Omron Sysmac Studio project DEMO_10 (Sysmac Studio 1.45.1.64010, StandardProject)

# Controller PLC: NX1P2-9024DT1 version 1.40
Task PrimaryTask (priority 4, period or condition 2000): Main_Prg
Library Mekatronik 1.0.0 (contents left out)

TYPE unW : UNION
    B : ARRAY[0..15] OF BOOL;
    BYT : ARRAY[0..1] OF BYTE;
    W : WORD;
END_UNION END_TYPE
TYPE unAlarm : UNION
    B : ARRAY[0..127] OF BOOL;
    LW : ARRAY[0..1] OF LWORD;
END_UNION END_TYPE
TYPE unUyari : UNION
    B : ARRAY[0..127] OF BOOL;
    LW : ARRAY[0..1] OF LWORD;
END_UNION END_TYPE
TYPE unTest : UNION
    B : ARRAY[0..127] OF BOOL;
    LW : ARRAY[0..1] OF LWORD;
END_UNION END_TYPE
TYPE ePLC_IO_St : STRUCT
    RealVars : ARRAY[1..64] OF REAL;  (* offset 0.0 *)
    IntegerVars : ARRAY[1..24] OF INT;  (* offset 256.0 *)
    String1_length : DINT;  (* offset 304.0 *)
    String1Var : STRING[82];  (* offset 308.0 *)
    String2_length : DINT;  (* offset 392.0 *)
    String2Var : STRING[82];  (* offset 396.0 *)
    SignalVars : ARRAY[1..64] OF BOOL;  (* offset 480.0 *)
END_STRUCT END_TYPE

VAR_GLOBAL
    From_Robot_C1 : ePLC_IO_St;  (* network input *)
    To_Robot_C1 : ePLC_IO_St;  (* network output *)
END_VAR

PROGRAM Main_Prg
VAR
    ToRo_Satrt : BOOL;
    FromRo_RobotAutoMode : BOOL;
    ytujty : REAL;
    ToRo_HareketModu : REAL;
    ToRo_IndexNumber : REAL;
    ToRo_PaletKat : REAL;
    FromRo_Haberlesme : BOOL;
    ToRo_Haberlesme : BOOL;
    konum_ok : BOOL;
    ToRo_x : REAL;
    ToRo_y : REAL;
    ToRo_z : REAL;
    ToRo_yaw : REAL;
    ToRo_pitch : REAL;
    ToRo_roll : REAL;
    izin : BOOL;
    ok : BOOL;
    campos : BOOL;
    campos1 : BOOL;
    konum1_ok : BOOL;
    ToRo_x1 : REAL;
    ToRo_y1 : REAL;
    ToRo_z1 : REAL;
    ToRo_yaw1 : REAL;
    ToRo_pitch1 : REAL;
    ToRo_roll1 : REAL;
END_VAR
VAR_EXTERNAL
    From_Robot_C1 : ePLC_IO_St;
    To_Robot_C1 : ePLC_IO_St;
END_VAR
VAR
    _e1 : R_TRIG;
    _e2 : R_TRIG;
    _e3 : R_TRIG;
    _e4 : R_TRIG;
END_VAR

(* Section Genel: ladder, written here as Structured Text *)

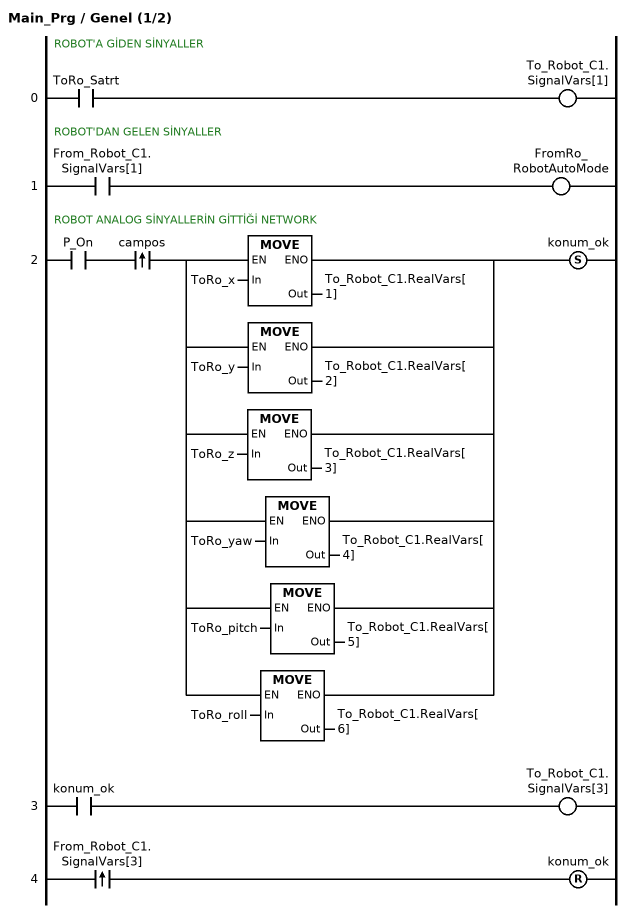
(* Rung 0: ROBOT'A GİDEN SİNYALLER *)
To_Robot_C1.SignalVars[1] := ToRo_Satrt;
(* Rung 1: ROBOT'DAN GELEN SİNYALLER *)
FromRo_RobotAutoMode := From_Robot_C1.SignalVars[1];
(* Rung 2: ROBOT ANALOG SİNYALLERİN GİTTİĞİ NETWORK *)
_e1(CLK := campos);
IF P_On AND _e1.Q THEN
    To_Robot_C1.RealVars[1] := ToRo_x;
    To_Robot_C1.RealVars[2] := ToRo_y;
    To_Robot_C1.RealVars[3] := ToRo_z;
    To_Robot_C1.RealVars[4] := ToRo_yaw;
    To_Robot_C1.RealVars[5] := ToRo_pitch;
    To_Robot_C1.RealVars[6] := ToRo_roll;
    konum_ok := TRUE;
END_IF;
(* Rung 3 *)
To_Robot_C1.SignalVars[3] := konum_ok;
(* Rung 4 *)
_e2(CLK := From_Robot_C1.SignalVars[3]);
IF _e2.Q THEN konum_ok := FALSE; END_IF;

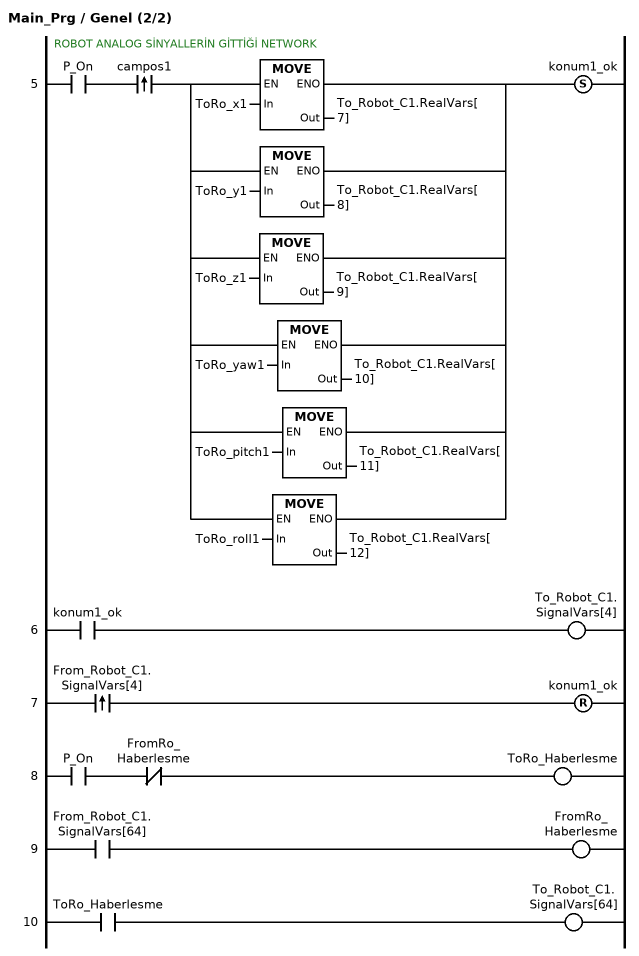
(* Rung 5: ROBOT ANALOG SİNYALLERİN GİTTİĞİ NETWORK *)
_e3(CLK := campos1);
IF P_On AND _e3.Q THEN
    To_Robot_C1.RealVars[7] := ToRo_x1;
    To_Robot_C1.RealVars[8] := ToRo_y1;
    To_Robot_C1.RealVars[9] := ToRo_z1;
    To_Robot_C1.RealVars[10] := ToRo_yaw1;
    To_Robot_C1.RealVars[11] := ToRo_pitch1;
    To_Robot_C1.RealVars[12] := ToRo_roll1;
    konum1_ok := TRUE;
END_IF;
(* Rung 6 *)
To_Robot_C1.SignalVars[4] := konum1_ok;
(* Rung 7 *)
_e4(CLK := From_Robot_C1.SignalVars[4]);
IF _e4.Q THEN konum1_ok := FALSE; END_IF;
(* Rung 8 *)
ToRo_Haberlesme := P_On AND NOT FromRo_Haberlesme;
(* Rung 9 *)
FromRo_Haberlesme := From_Robot_C1.SignalVars[64];
(* Rung 10 *)
To_Robot_C1.SignalVars[64] := ToRo_Haberlesme;
END_PROGRAM

FUNCTION_BLOCK myHome_FB
VAR
    MC_SetPosition_Homming : MC_SetPosition;
    MC_MoveAbsolute_Homming : MC_MoveAbsolute;
    Step_Home : INT;
    MC_MoveVelocity_1 : MC_MoveVelocity;
    TON_5 : TON;
    TON_6 : TON;
    MC_MoveVelocity_2 : MC_MoveVelocity;
    MC_MoveVelocity_11 : MC_MoveVelocity;
    MC_MoveVelocity_12 : MC_MoveVelocity;
    TP_1 : TP;
    TON_1 : TON;
    TON_2 : TON;
    Stop_Axis_1 : BOOL;
    Stop_Axis_2 : BOOL;
    HomePositionSensorInternal : LREAL;
    MC_Stop_Homming1 : MC_Stop;
    MC_Stop_Homming2 : MC_Stop;
    InPlaceHomed : BOOL;
    tr : BOOL;
    tr1 : BOOL;
END_VAR
VAR_IN_OUT CONSTANT
    Axis : _sAXIS_REF;
END_VAR
VAR_INPUT
    Start_Homming : BOOL;
    Direction : BOOL;
    ReverseDown : BOOL;
    UP_DN : BOOL;
    InPlace : BOOL;
    Home_Sensor : BOOL;
    EMG : BOOL;
    Stop : BOOL;
    HomeSpeed : LREAL;
    HomeSpeedLow : LREAL;
    OffsetPosition : LREAL;
    HomeSensorPosition : LREAL;
    ResetHomeOK : BOOL;
    IleriLimit : BOOL;
    GeriLimit : BOOL;
    Acceleration : LREAL;
    Deceleration : LREAL;
END_VAR
VAR_OUTPUT
    Home_Ok : BOOL;
    Busy : BOOL;
    Error : BOOL;
    LimitsError : BOOL;
END_VAR
VAR
    _e1 : R_TRIG;
    _p2 : BOOL;
    _p3 : BOOL;
    _br13_0 : BOOL;
    _br13_1 : BOOL;
    _br13_2 : BOOL;
    _e4 : R_TRIG;
    _e5 : R_TRIG;
    _e6 : R_TRIG;
    _e7 : F_TRIG;
    _br17_0 : BOOL;
    _br17_1 : BOOL;
    _br17_2 : BOOL;
    _e8 : R_TRIG;
END_VAR
(* ladder, written here as Structured Text *)

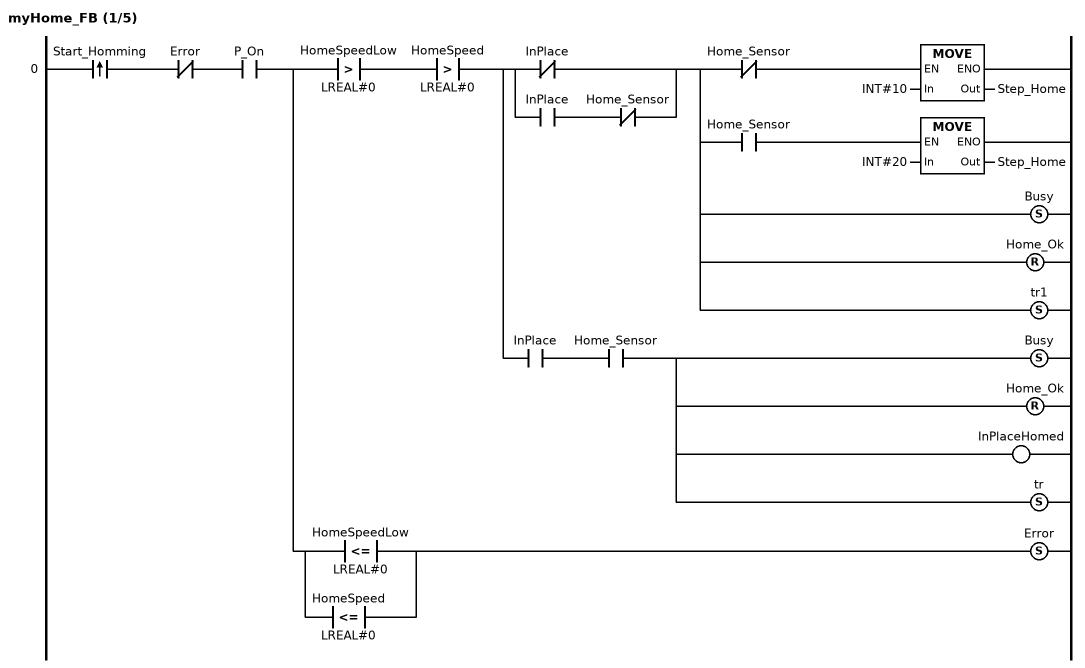
(* Rung 0 *)
_e1(CLK := Start_Homming);
_p2 := _e1.Q AND NOT Error AND P_On AND (HomeSpeedLow > LREAL#0) AND (HomeSpeed > LREAL#0);
_p3 := _p2 AND (NOT InPlace OR (InPlace AND NOT Home_Sensor));
IF _p3 AND NOT Home_Sensor THEN Step_Home := INT#10; END_IF;
IF _p3 AND Home_Sensor THEN Step_Home := INT#20; END_IF;
IF _p3 THEN
    Busy := TRUE;
    Home_Ok := FALSE;
    tr1 := TRUE;
END_IF;
IF _p2 AND InPlace AND Home_Sensor THEN
    Busy := TRUE;
    Home_Ok := FALSE;
END_IF;
InPlaceHomed := _p2 AND InPlace AND Home_Sensor;
IF _p2 AND InPlace AND Home_Sensor THEN tr := TRUE; END_IF;
IF _e1.Q AND NOT Error AND P_On AND ((HomeSpeedLow <= LREAL#0) OR (HomeSpeed <= LREAL#0)) THEN
    Error := TRUE;
END_IF;

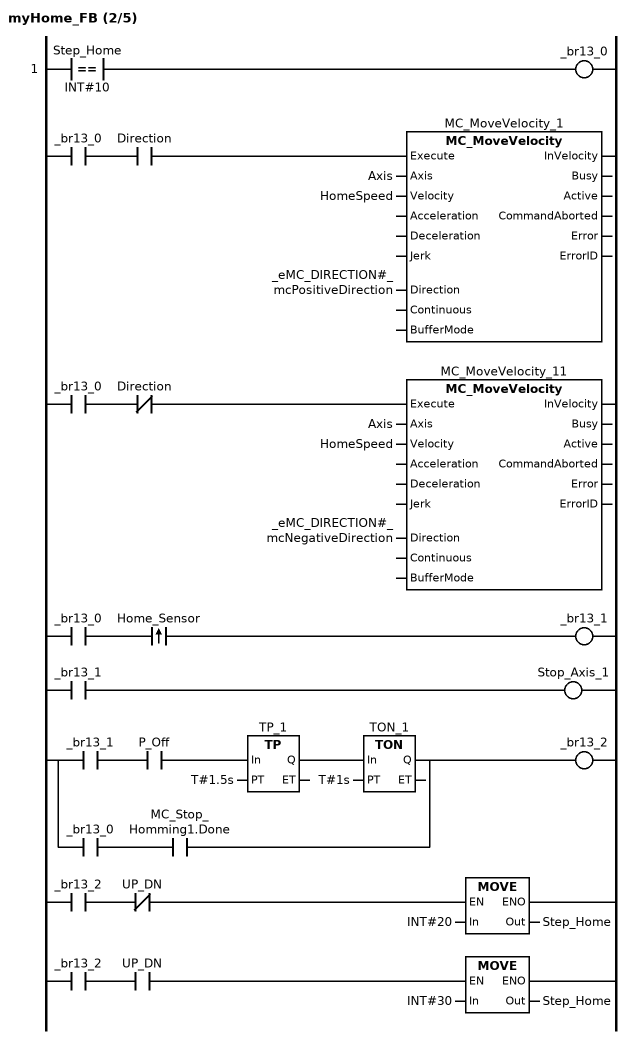
(* Rung 1 *)
_br13_0 := Step_Home = INT#10;
MC_MoveVelocity_1(Execute := _br13_0 AND Direction, Axis := Axis, Velocity := HomeSpeed, Direction := _eMC_DIRECTION#_mcPositiveDirection);
MC_MoveVelocity_11(Execute := _br13_0 AND NOT Direction, Axis := Axis, Velocity := HomeSpeed, Direction := _eMC_DIRECTION#_mcNegativeDirection);
_e4(CLK := Home_Sensor);
_br13_1 := _br13_0 AND _e4.Q;
Stop_Axis_1 := _br13_1;
TP_1(In := _br13_1 AND P_Off, PT := T#1.5s);
TON_1(In := TP_1.Q, PT := T#1s);
_br13_2 := TON_1.Q OR (_br13_0 AND MC_Stop_Homming1.Done);
IF _br13_2 AND NOT UP_DN THEN Step_Home := INT#20; END_IF;
IF _br13_2 AND UP_DN THEN Step_Home := INT#30; END_IF;

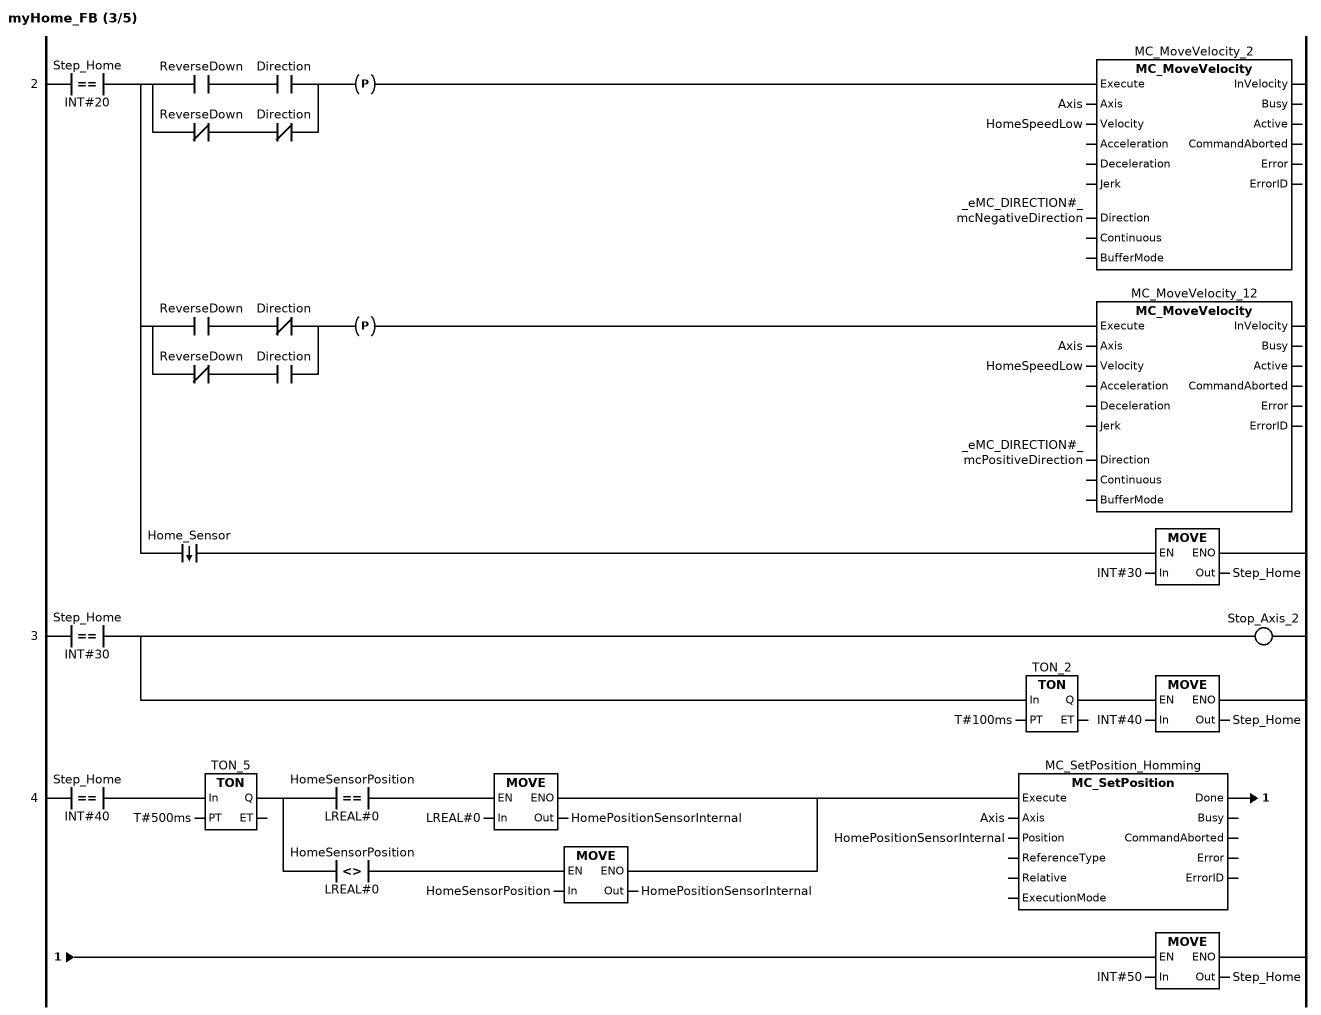
(* Rung 2 *)
_e5(CLK := (Step_Home = INT#20) AND ((ReverseDown AND Direction) OR (NOT ReverseDown AND NOT Direction)));
MC_MoveVelocity_2(Execute := _e5.Q, Axis := Axis, Velocity := HomeSpeedLow, Direction := _eMC_DIRECTION#_mcNegativeDirection);
_e6(CLK := (Step_Home = INT#20) AND ((ReverseDown AND NOT Direction) OR (NOT ReverseDown AND Direction)));
MC_MoveVelocity_12(Execute := _e6.Q, Axis := Axis, Velocity := HomeSpeedLow, Direction := _eMC_DIRECTION#_mcPositiveDirection);
_e7(CLK := Home_Sensor);
IF (Step_Home = INT#20) AND _e7.Q THEN Step_Home := INT#30; END_IF;
(* Rung 3 *)
Stop_Axis_2 := Step_Home = INT#30;
TON_2(In := Step_Home = INT#30, PT := T#100ms);
IF TON_2.Q THEN Step_Home := INT#40; END_IF;
(* Rung 4 *)
TON_5(In := Step_Home = INT#40, PT := T#500ms);
IF TON_5.Q AND (HomeSensorPosition = LREAL#0) THEN HomePositionSensorInternal := LREAL#0; END_IF;
IF TON_5.Q AND (HomeSensorPosition <> LREAL#0) THEN
    HomePositionSensorInternal := HomeSensorPosition;
END_IF;
MC_SetPosition_Homming(Execute := TON_5.Q AND ((HomeSensorPosition = LREAL#0) OR (HomeSensorPosition <> LREAL#0)), Axis := Axis, Position := HomePositionSensorInternal);
IF MC_SetPosition_Homming.Done THEN Step_Home := INT#50; END_IF;

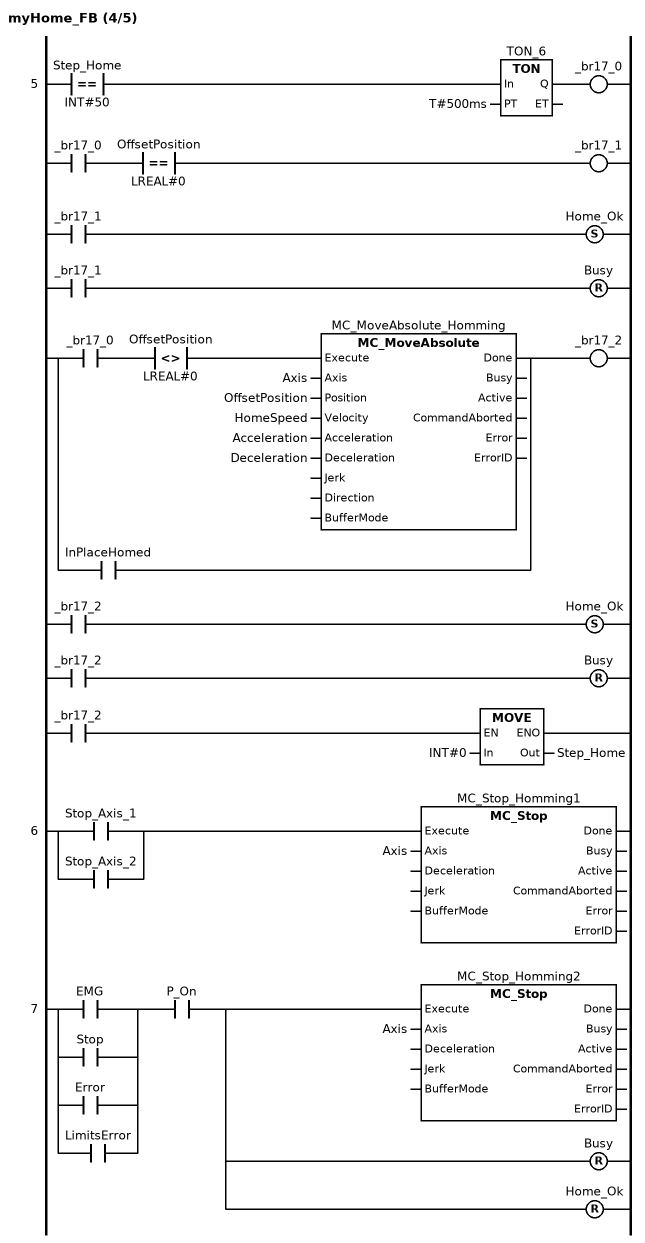
(* Rung 5 *)
TON_6(In := Step_Home = INT#50, PT := T#500ms);
_br17_0 := TON_6.Q;
_br17_1 := _br17_0 AND (OffsetPosition = LREAL#0);
IF _br17_1 THEN Home_Ok := TRUE; END_IF;
IF _br17_1 THEN Busy := FALSE; END_IF;
MC_MoveAbsolute_Homming(Execute := _br17_0 AND (OffsetPosition <> LREAL#0), Axis := Axis, Position := OffsetPosition, Velocity := HomeSpeed, Acceleration := Acceleration, Deceleration := Deceleration);
_br17_2 := MC_MoveAbsolute_Homming.Done OR InPlaceHomed;
IF _br17_2 THEN Home_Ok := TRUE; END_IF;
IF _br17_2 THEN Busy := FALSE; END_IF;
IF _br17_2 THEN Step_Home := INT#0; END_IF;
(* Rung 6 *)
MC_Stop_Homming1(Execute := Stop_Axis_1 OR Stop_Axis_2, Axis := Axis);
(* Rung 7 *)
MC_Stop_Homming2(Execute := (EMG OR Stop OR Error OR LimitsError) AND P_On, Axis := Axis);
IF (EMG OR Stop OR Error OR LimitsError) AND P_On THEN
    Busy := FALSE;
    Home_Ok := FALSE;
END_IF;

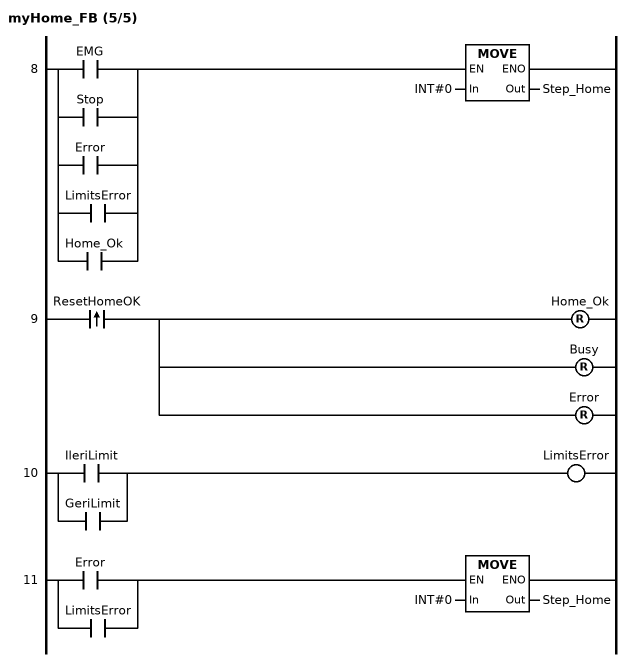
(* Rung 8 *)
IF EMG OR Stop OR Error OR LimitsError OR Home_Ok THEN Step_Home := INT#0; END_IF;
(* Rung 9 *)
_e8(CLK := ResetHomeOK);
IF _e8.Q THEN
    Home_Ok := FALSE;
    Busy := FALSE;
    Error := FALSE;
END_IF;
(* Rung 10 *)
LimitsError := IleriLimit OR GeriLimit;
(* Rung 11 *)
IF Error OR LimitsError THEN Step_Home := INT#0; END_IF;
END_FUNCTION_BLOCK

FUNCTION_BLOCK myHomeV2_FB
VAR
    MC_SetPosition_Homming : MC_SetPosition;
    MC_MoveAbsolute_Homming : MC_MoveAbsolute;
    Step_Home : INT;
    MC_MoveVelocity_1 : MC_MoveVelocity;
    TON_6 : TON;
    MC_MoveVelocity_2 : MC_MoveVelocity;
    MC_MoveVelocity_11 : MC_MoveVelocity;
    MC_MoveVelocity_12 : MC_MoveVelocity;
    TON_1 : TON;
    Stop_Axis_1 : BOOL;
    Stop_Axis_2 : BOOL;
    HomePositionSensorInternal : LREAL;
    MC_Stop_Homming1 : MC_Stop;
    MC_Stop_Homming2 : MC_Stop;
    InPlaceHomed : BOOL;
    Stop_Axis_Done : BOOL;
    Busy1 : BOOL;
    Busy2 : BOOL;
END_VAR
VAR_IN_OUT CONSTANT
    Axis : _sAXIS_REF;
END_VAR
VAR_INPUT
    Start_Homming : BOOL;
    Direction : BOOL;
    ReverseDown : BOOL;
    UP_DN : BOOL;
    InPlace : BOOL;
    Home_Sensor : BOOL;
    EMG : BOOL;
    Stop : BOOL;
    HomeSpeed : LREAL;
    HomeSpeedLow : LREAL;
    OffsetPosition : LREAL;
    HomeSensorPosition : LREAL;
    ResetHomeOK : BOOL;
    IleriLimit : BOOL;
    GeriLimit : BOOL;
    Acceleration : LREAL;
    Deceleration : LREAL;
END_VAR
VAR_OUTPUT
    Home_Ok : BOOL;
    Busy : BOOL;
    Error : BOOL;
    LimitsError : BOOL;
END_VAR
VAR
    _e1 : R_TRIG;
    _p2 : BOOL;
    _p3 : BOOL;
    _e4 : R_TRIG;
    _e5 : R_TRIG;
    _p6 : BOOL;
    _e7 : F_TRIG;
    _br30_0 : BOOL;
    _br30_1 : BOOL;
    _br30_2 : BOOL;
    _e8 : R_TRIG;
END_VAR
(* ladder, written here as Structured Text *)

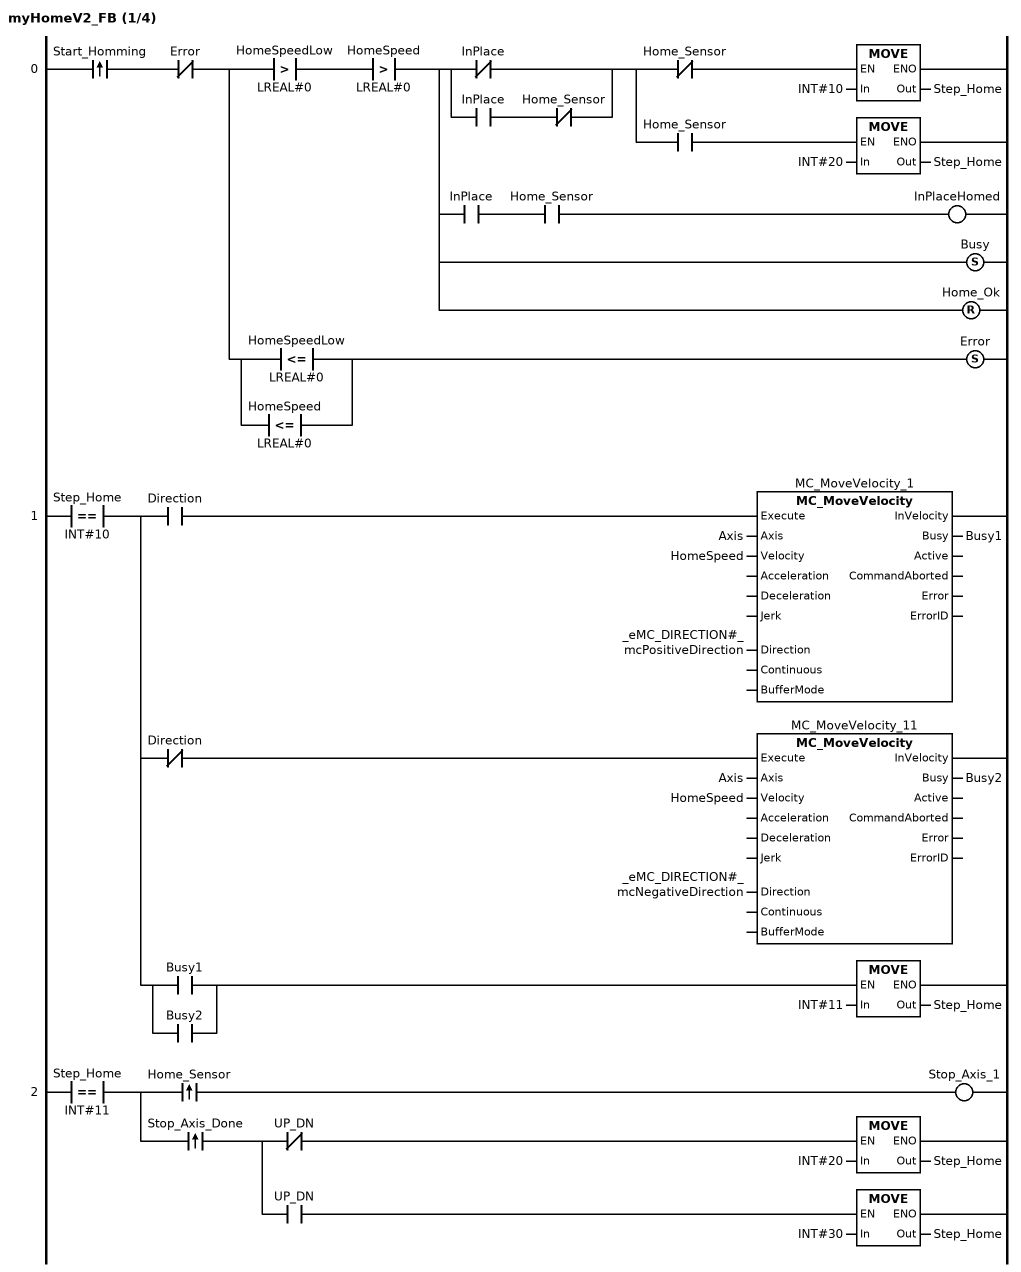
(* Rung 0 *)
_e1(CLK := Start_Homming);
_p2 := _e1.Q AND NOT Error AND (HomeSpeedLow > LREAL#0) AND (HomeSpeed > LREAL#0);
_p3 := _p2 AND (NOT InPlace OR (InPlace AND NOT Home_Sensor));
IF _p3 AND NOT Home_Sensor THEN Step_Home := INT#10; END_IF;
IF _p3 AND Home_Sensor THEN Step_Home := INT#20; END_IF;
InPlaceHomed := _p2 AND InPlace AND Home_Sensor;
IF _p2 THEN
    Busy := TRUE;
    Home_Ok := FALSE;
END_IF;
IF _e1.Q AND NOT Error AND ((HomeSpeedLow <= LREAL#0) OR (HomeSpeed <= LREAL#0)) THEN
    Error := TRUE;
END_IF;
(* Rung 1 *)
MC_MoveVelocity_1(Execute := (Step_Home = INT#10) AND Direction, Axis := Axis, Velocity := HomeSpeed, Direction := _eMC_DIRECTION#_mcPositiveDirection, Busy => Busy1);
MC_MoveVelocity_11(Execute := (Step_Home = INT#10) AND NOT Direction, Axis := Axis, Velocity := HomeSpeed, Direction := _eMC_DIRECTION#_mcNegativeDirection, Busy => Busy2);
IF (Step_Home = INT#10) AND (Busy1 OR Busy2) THEN Step_Home := INT#11; END_IF;
(* Rung 2 *)
_e4(CLK := Home_Sensor);
Stop_Axis_1 := (Step_Home = INT#11) AND _e4.Q;
_e5(CLK := Stop_Axis_Done);
_p6 := (Step_Home = INT#11) AND _e5.Q;
IF (Step_Home = INT#11) AND _e5.Q AND NOT UP_DN THEN Step_Home := INT#20; END_IF;
IF _p6 AND UP_DN THEN Step_Home := INT#30; END_IF;

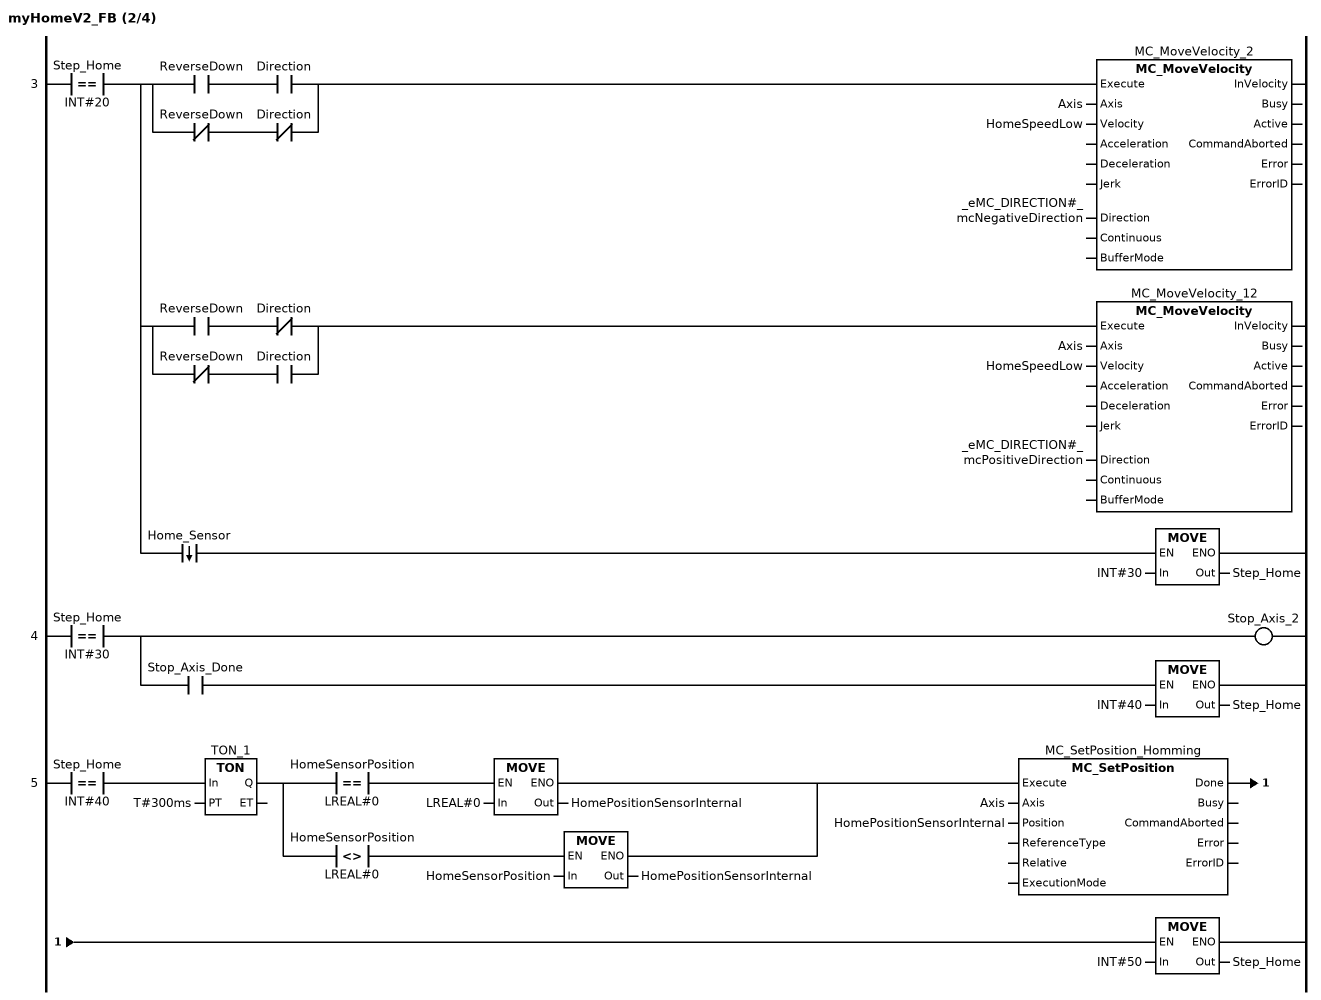
(* Rung 3 *)
MC_MoveVelocity_2(Execute := (Step_Home = INT#20) AND ((ReverseDown AND Direction) OR (NOT ReverseDown AND NOT Direction)), Axis := Axis, Velocity := HomeSpeedLow, Direction := _eMC_DIRECTION#_mcNegativeDirection);
MC_MoveVelocity_12(Execute := (Step_Home = INT#20) AND ((ReverseDown AND NOT Direction) OR (NOT ReverseDown AND Direction)), Axis := Axis, Velocity := HomeSpeedLow, Direction := _eMC_DIRECTION#_mcPositiveDirection);
_e7(CLK := Home_Sensor);
IF (Step_Home = INT#20) AND _e7.Q THEN Step_Home := INT#30; END_IF;
(* Rung 4 *)
Stop_Axis_2 := Step_Home = INT#30;
IF (Step_Home = INT#30) AND Stop_Axis_Done THEN Step_Home := INT#40; END_IF;
(* Rung 5 *)
TON_1(In := Step_Home = INT#40, PT := T#300ms);
IF TON_1.Q AND (HomeSensorPosition = LREAL#0) THEN HomePositionSensorInternal := LREAL#0; END_IF;
IF TON_1.Q AND (HomeSensorPosition <> LREAL#0) THEN
    HomePositionSensorInternal := HomeSensorPosition;
END_IF;
MC_SetPosition_Homming(Execute := TON_1.Q AND ((HomeSensorPosition = LREAL#0) OR (HomeSensorPosition <> LREAL#0)), Axis := Axis, Position := HomePositionSensorInternal);
IF MC_SetPosition_Homming.Done THEN Step_Home := INT#50; END_IF;

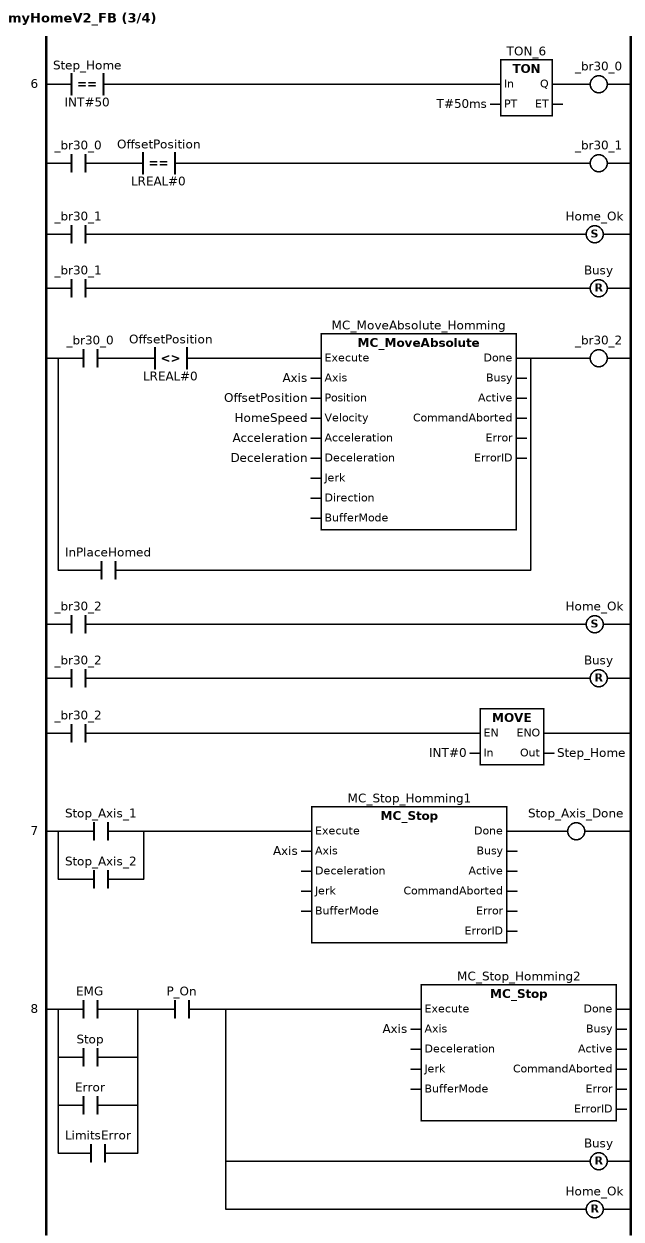
(* Rung 6 *)
TON_6(In := Step_Home = INT#50, PT := T#50ms);
_br30_0 := TON_6.Q;
_br30_1 := _br30_0 AND (OffsetPosition = LREAL#0);
IF _br30_1 THEN Home_Ok := TRUE; END_IF;
IF _br30_1 THEN Busy := FALSE; END_IF;
MC_MoveAbsolute_Homming(Execute := _br30_0 AND (OffsetPosition <> LREAL#0), Axis := Axis, Position := OffsetPosition, Velocity := HomeSpeed, Acceleration := Acceleration, Deceleration := Deceleration);
_br30_2 := MC_MoveAbsolute_Homming.Done OR InPlaceHomed;
IF _br30_2 THEN Home_Ok := TRUE; END_IF;
IF _br30_2 THEN Busy := FALSE; END_IF;
IF _br30_2 THEN Step_Home := INT#0; END_IF;
(* Rung 7 *)
MC_Stop_Homming1(Execute := Stop_Axis_1 OR Stop_Axis_2, Axis := Axis);
Stop_Axis_Done := MC_Stop_Homming1.Done;
(* Rung 8 *)
MC_Stop_Homming2(Execute := (EMG OR Stop OR Error OR LimitsError) AND P_On, Axis := Axis);
IF (EMG OR Stop OR Error OR LimitsError) AND P_On THEN
    Busy := FALSE;
    Home_Ok := FALSE;
END_IF;

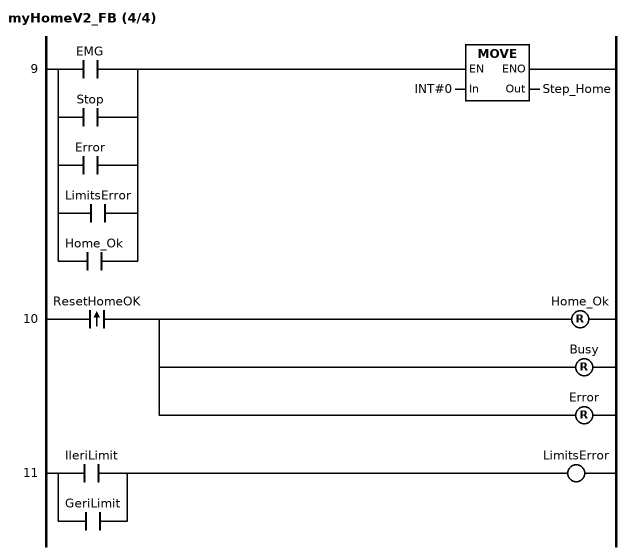
(* Rung 9 *)
IF EMG OR Stop OR Error OR LimitsError OR Home_Ok THEN Step_Home := INT#0; END_IF;
(* Rung 10 *)
_e8(CLK := ResetHomeOK);
IF _e8.Q THEN
    Home_Ok := FALSE;
    Busy := FALSE;
    Error := FALSE;
END_IF;
(* Rung 11 *)
LimitsError := IleriLimit OR GeriLimit;
END_FUNCTION_BLOCK